// Global variables for the TraceTek leak detector
{attribute 'qualified_only'}
VAR_GLOBAL CONSTANT
    (* Modbus address *)
    nModbusSlaveAddress : BYTE := 199; // Modbus slave address of the TraceTek device
END_VAR
VAR_GLOBAL PERSISTENT
    {attribute 'pytmc' := 'pv: @(BASE):LPS:LEAK'}
    stLeakMonitorBoundaries : ST_LeakBoundaries; // Boundaries of possible leak locations
END_VAR

(* stored: Version 1.1.0.1, ProductVersion 3.1.4022.18
   GVL GVL_TraceTek: Id {69094c0a-8e7d-4944-912b-7a8aa3ff193d} *)
